FUNCTION_BLOCK testDNC1 (* Composite Function Block Type *)
  (* Standard: 61499-2 *)
  (* Version 0.0, 2015-11-12, 4DIAC-IDE, 4DIAC-Consortium *)
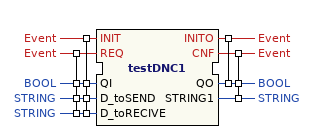
  EVENT_INPUT
    INIT WITH QI, D_toSEND, D_toRECIVE; (* Initialization Request *)
    REQ WITH QI, D_toSEND, D_toRECIVE; (* Normal Execution Request *)
  END_EVENT
  EVENT_OUTPUT
    INITO WITH QO; (* Initialization Confirm *)
    CNF WITH QO, STRING1; (* Execution Confirmation *)
  END_EVENT
  VAR_INPUT
    QI : BOOL; (* Input event qualifier *)
    D_toSEND : STRING;
    D_toRECIVE : STRING;
  END_VAR
  VAR_OUTPUT
    QO : BOOL; (* Output event qualifier *)
    STRING1 : STRING;
  END_VAR
  FBS
    F_NOT_1_0 : F_NOT;
    BASIC_SEND_ENQ_1_0_0 : BASIC_SEND_ENQ;
    SIFB_RAWSTRING_EQ_0_0_0 : SIFB_RAWSTRING_EQ;
    E_MERGE_2_0 : E_MERGE;
    E_PERMIT_1_1_0_0_1 : E_PERMIT;
    E_MERGE_2_1 : E_MERGE;
    E_SPLIT_1_0_0 : E_SPLIT;
    E_SPLIT_1_1_0 : E_SPLIT;
    E_SPLIT_1_2 : E_SPLIT;
    E_CTU_0 : E_CTU(PV := 0);
    B_DEMUX_BOOL_0 : B_DEMUX_BOOL;
    E_MERGE_2 : E_MERGE;
    E_PERMIT_1_3 : E_PERMIT;
    E_DELAY_0 : E_DELAY(DT := T#10s);
    E_PERMIT_1_1_0_0_0 : E_PERMIT;
    BASIC_SEND_ENQ_1_0 : BASIC_SEND_ENQ;
    STRING_SPLIT_0 : STRING_SPLIT;
    E_SPLIT_1_0_0_0 : E_SPLIT;
    E_SPLIT_1_1_0_1 : E_SPLIT;
    E_PERMIT_1_0_1_0 : E_PERMIT;
    E_SR_1 : E_SR;
    F_LE_0 : F_LE(IN2 := UINT#2);
    E_MERGE_1_0 : E_MERGE;
    E_SPLIT_1_1_0_1_0 : E_SPLIT;
    E_DELAY_0_0 : E_DELAY(DT := T#100ms);
    SIFB_RAWSTRING_EQ_0_0 : SIFB_RAWSTRING_EQ;
    STRING2STRING_1 : STRING2STRING;
    E_SR_1_0 : E_SR;
    F_NOT_1 : F_NOT;
    E_SPLIT_1_0 : E_SPLIT;
    E_PERMIT_1_3_0 : E_PERMIT;
    E_MERGE_1 : E_MERGE;
    BASIC_SEND_EOT_1 : BASIC_SEND_EOT;
    STRING_SPLIT_0_0 : STRING_SPLIT;
    STRING2STRING_1_1_0 : STRING2STRING;
    E_CTU_0_0 : E_CTU(PV := 0);
    E_PERMIT_1_1_0_1_0 : E_PERMIT;
    E_PERMIT_1_1_0_1 : E_PERMIT;
    E_SPLIT_1_1 : E_SPLIT;
    E_SPLIT_1_1_0_0 : E_SPLIT;
    E_SPLIT_1 : E_SPLIT;
    E_MERGE_0 : E_MERGE;
    F_NOT_1_0_1 : F_NOT;
    E_PERMIT_1_0_1 : E_PERMIT;
    CLIENT_1_0 : CLIENT_1(QI := BOOL#1, ID := ser[COM3]);
    BASIC_SEND_NAKDEL_1 : BASIC_SEND_NAKDEL;
    E_PERMIT_1_1_0_0 : E_PERMIT;
    F_NOT_1_0_0 : F_NOT;
    E_PERMIT_1_1_0_0_0_0 : E_PERMIT;
    E_MERGE_3 : E_MERGE;
    E_PERMIT_1_1_0 : E_PERMIT;
    F_LE_0_0 : F_LE(IN2 := UINT#2);
    STRING2STRING_1_1_0_1 : STRING2STRING;
    STRING2STRING_1_1_0_1_1 : STRING2STRING;
  END_FBS
  EVENT_CONNECTIONS
    B_DEMUX_BOOL_0.CNF TO E_PERMIT_1_1_0_0_0_0.EI;
    E_DELAY_0.EO TO E_MERGE_1_0.EI2;
    E_SPLIT_1_1_0_0.EO2 TO E_CTU_0.R;
    E_CTU_0.CUO TO F_LE_0.REQ;
    E_PERMIT_1_0_1.EO TO E_MERGE_0.EI1;
    F_NOT_1_0_1.CNF TO E_PERMIT_1_1_0_0_1.EI;
    E_MERGE_2_1.EO TO E_DELAY_0.START;
    E_MERGE_1.EO TO E_SPLIT_1_0.EI;
    E_PERMIT_1_1_0_1.EO TO CLIENT_1_0.REQ;
    E_SPLIT_1_1_0.EO2 TO E_CTU_0_0.R;
    BASIC_SEND_ENQ_1_0_0.EO TO STRING2STRING_1_1_0.REQ;
    E_SPLIT_1_0_0_0.EO2 TO E_MERGE_2_0.EI2;
    E_SPLIT_1.EO2 TO STRING2STRING_1.REQ;
    E_SPLIT_1_1_0.EO1 TO E_SPLIT_1_1_0_0.EI;
    E_SPLIT_1_1.EO2 TO E_PERMIT_1_1_0_0.EI;
    E_SPLIT_1_2.EO2 TO B_DEMUX_BOOL_0.EI2;
    SIFB_RAWSTRING_EQ_0_0_0.EO TO E_SPLIT_1_1.EI;
    F_NOT_1.CNF TO E_PERMIT_1_0_1.EI;
    E_SPLIT_1_0_0_0.EO1 TO STRING_SPLIT_0.EI3;
    E_SPLIT_1_1_0_0.EO1 TO E_MERGE_2.EI2;
    E_PERMIT_1_1_0_1_0.EO TO SIFB_RAWSTRING_EQ_0_0.EI;
    E_SPLIT_1_0.EO1 TO E_MERGE_2_1.EI1;
    BASIC_SEND_ENQ_1_0.EO TO STRING_SPLIT_0.EI2;
    STRING_SPLIT_0.EO TO E_PERMIT_1_1_0_1.EI;
    E_SPLIT_1_1_0_1.EO1 TO E_CTU_0_0.CU;
    E_PERMIT_1_3.EO TO E_MERGE_1.EI1;
    E_PERMIT_1_1_0_0_0_0.EO TO BASIC_SEND_ENQ_1_0.EI;
    E_CTU_0_0.CUO TO F_LE_0_0.REQ;
    F_LE_0_0.CNF TO F_NOT_1_0.REQ;
    SIFB_RAWSTRING_EQ_0_0.EO TO BASIC_SEND_NAKDEL_1.REQ;
    E_SPLIT_1_0.EO2 TO B_DEMUX_BOOL_0.EI1;
    E_MERGE_2_0.EO TO E_DELAY_0_0.START;
    E_SPLIT_1.EO1 TO E_MERGE_2_1.EI2;
    E_PERMIT_1_1_0_0_0.EO TO F_NOT_1_0_1.REQ;
    E_MERGE_3.EO TO E_SPLIT_1.EI;
    STRING2STRING_1.CNF TO STRING_SPLIT_0.EI1;
    E_PERMIT_1_1_0_0_1.EO TO E_MERGE_1_0.EI1;
    F_NOT_1_0.CNF TO E_SPLIT_1_1_0_1_0.EI;
    E_PERMIT_1_0_1_0.EO TO E_MERGE_0.EI2;
    F_LE_0.CNF TO F_NOT_1.REQ;
    STRING_SPLIT_0_0.EO TO E_PERMIT_1_1_0_1_0.EI;
    E_PERMIT_1_3_0.EO TO E_MERGE_3.EI2;
    BASIC_SEND_NAKDEL_1.CNF TO SIFB_RAWSTRING_EQ_0_0_0.EI;
    CLIENT_1_0.INITO TO BASIC_SEND_ENQ_1_0_0.EI;
    E_SR_1_0.EO TO E_SPLIT_1_2.EI;
    E_PERMIT_1_1_0.EO TO E_SPLIT_1_1_0.EI;
    E_SPLIT_1_0_0.EO2 TO E_MERGE_2_0.EI1;
    E_SPLIT_1_0_0.EO1 TO STRING_SPLIT_0.EI4;
    E_DELAY_0_0.EO TO E_SR_1.R;
    E_MERGE_0.EO TO BASIC_SEND_EOT_1.REQ;
    E_SPLIT_1_2.EO3 TO E_SR_1.S;
    E_SPLIT_1_1_0_1_0.EO2 TO E_PERMIT_1_0_1_0.EI;
    E_MERGE_1_0.EO TO E_CTU_0.CU;
    F_NOT_1_0_0.CNF TO E_PERMIT_1_1_0_0_0.EI;
    E_SPLIT_1_1_0_1.EO2 TO E_MERGE_2.EI1;
    F_LE_0.CNF TO E_PERMIT_1_3.EI;
    E_SPLIT_1_1_0_1_0.EO1 TO E_PERMIT_1_3_0.EI;
    E_PERMIT_1_1_0_0.EO TO E_SPLIT_1_1_0_1.EI;
    BASIC_SEND_EOT_1.CNF TO E_SPLIT_1_0_0_0.EI;
    E_SPLIT_1_1.EO1 TO E_PERMIT_1_1_0.EI;
    E_MERGE_2.EO TO E_DELAY_0.STOP;
    CLIENT_1_0.CNF TO STRING_SPLIT_0_0.EI1;
    E_SPLIT_1_1.EO3 TO F_NOT_1_0_0.REQ;
    REQ TO E_MERGE_3.EI1;
    INIT TO CLIENT_1_0.INIT;
    STRING2STRING_1_1_0.CNF TO STRING2STRING_1_1_0_1.REQ;
    STRING2STRING_1_1_0_1.CNF TO E_SR_1_0.S;
    E_SPLIT_1_1_0.EO3 TO E_SPLIT_1_0_0.EI;
    E_SPLIT_1_0_0.EO3 TO STRING2STRING_1_1_0_1_1.REQ;
    STRING2STRING_1_1_0_1_1.CNF TO CNF;
    E_SPLIT_1_2.EO1 TO INITO;
  END_CONNECTIONS
  DATA_CONNECTIONS
    E_CTU_0.CV TO F_LE_0.IN1;
    F_NOT_1.OUT TO E_PERMIT_1_0_1.PERMIT;
    E_SR_1.Q TO E_PERMIT_1_1_0_1.PERMIT;
    F_LE_0.OUT TO F_NOT_1.IN;
    SIFB_RAWSTRING_EQ_0_0_0.OUT TO F_NOT_1_0_0.IN;
    STRING2STRING_1.OUT TO STRING_SPLIT_0.STRING1;
    F_NOT_1_0_0.OUT TO E_PERMIT_1_1_0_0_0.PERMIT;
    E_SR_1.Q TO E_PERMIT_1_1_0_1_0.PERMIT;
    BASIC_SEND_EOT_1.OUT TO STRING_SPLIT_0.STRING3;
    SIFB_RAWSTRING_EQ_0_0_0.OUT TO E_PERMIT_1_1_0_0.PERMIT;
    SIFB_RAWSTRING_EQ_0_0.OUT TO F_NOT_1_0_1.IN;
    SIFB_RAWSTRING_EQ_0_0.OUT TO E_PERMIT_1_1_0.PERMIT;
    F_NOT_1_0.OUT TO E_PERMIT_1_0_1_0.PERMIT;
    STRING_SPLIT_0.OUT TO CLIENT_1_0.SD_1;
    CLIENT_1_0.RD_1 TO STRING_SPLIT_0_0.STRING1;
    STRING_SPLIT_0_0.OUT TO SIFB_RAWSTRING_EQ_0_0.IN1;
    F_NOT_1_0_1.OUT TO E_PERMIT_1_1_0_0_1.PERMIT;
    STRING_SPLIT_0_0.OUT TO SIFB_RAWSTRING_EQ_0_0_0.IN1;
    F_LE_0.OUT TO B_DEMUX_BOOL_0.IN1;
    F_LE_0.OUT TO E_PERMIT_1_3.PERMIT;
    E_SR_1_0.Q TO B_DEMUX_BOOL_0.IN2;
    E_CTU_0_0.CV TO F_LE_0_0.IN1;
    B_DEMUX_BOOL_0.OUT TO E_PERMIT_1_1_0_0_0_0.PERMIT;
    F_LE_0_0.OUT TO F_NOT_1_0.IN;
    F_LE_0_0.OUT TO E_PERMIT_1_3_0.PERMIT;
    STRING2STRING_1_1_0.OUT TO STRING2STRING_1.IN;
    BASIC_SEND_ENQ_1_0.OUT TO STRING_SPLIT_0.STRING2;
    BASIC_SEND_NAKDEL_1.OUT TO SIFB_RAWSTRING_EQ_0_0_0.IN2;
    D_toSEND TO STRING2STRING_1_1_0.IN;
    STRING2STRING_1_1_0_1.OUT TO SIFB_RAWSTRING_EQ_0_0.IN2;
    D_toRECIVE TO STRING2STRING_1_1_0_1.IN;
    STRING_SPLIT_0_0.OUT TO STRING2STRING_1_1_0_1_1.IN;
    STRING2STRING_1_1_0_1_1.OUT TO STRING1;
  END_CONNECTIONS
END_FUNCTION_BLOCK
